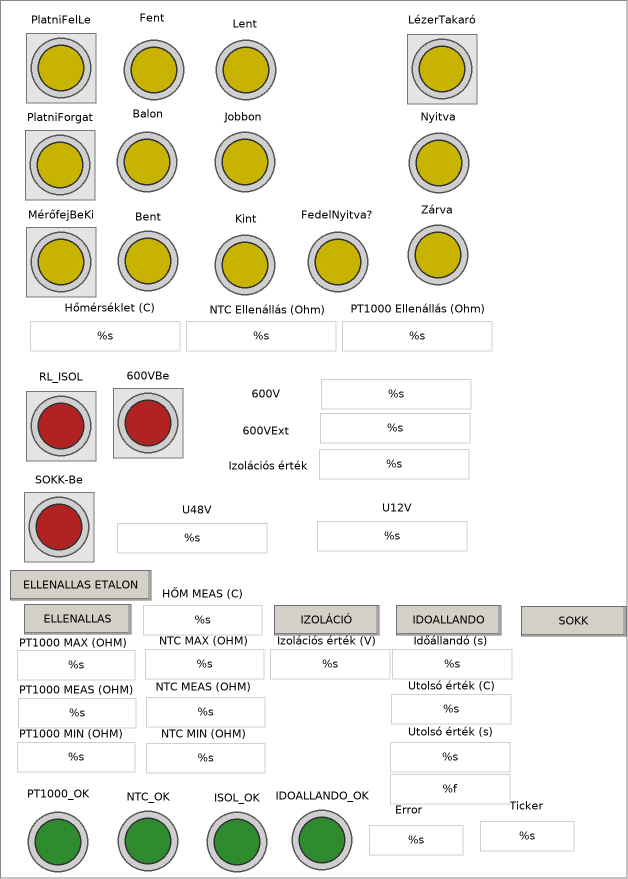
VISUALIZATION TempPistiVegmero  // 628x879
    Lamp1 (211,35 70x70), variable: VEGMERO.bPlatniLent, style: Lamp-Lamp1-Yellow
    Label (190,9 110x30), "Lent"
    PushSwitch (26,33 70x70), variable: VEGMERO.bPlatniFelLe, behaviour: TOGGLE, style: Switch-PushSwitch-Yellow
    Label (6,5 110x30), "PlatniFelLe"
    Lamp1 (112,127 70x70), variable: VEGMERO.bPlatniBalon, style: Lamp-Lamp1-Yellow
    Label (93,99 110x30), "Balon"
    Lamp1 (210,127 70x70), variable: VEGMERO.bPlatniJobbon, style: Lamp-Lamp1-Yellow
    Label (188,102 110x30), "Jobbon"
    PushSwitch (25,130 70x70), variable: VEGMERO.bPlatniBalraJobbra, behaviour: TOGGLE, style: Switch-PushSwitch-Yellow
    Label (5,103 110x29), "PlatniForgat"
    Lamp1 (113,226 70x70), variable: VEGMERO.bMerotukBent, style: Lamp-Lamp1-Yellow
    Label (93,202 110x30), "Bent"
    Lamp1 (210,230 70x70), variable: VEGMERO.bMerotukKint, style: Lamp-Lamp1-Yellow
    Label (191,204 110x30), "Kint"
    PushSwitch (26,227 70x70), variable: VEGMERO.bMerotukBeKi, behaviour: TOGGLE, style: Switch-PushSwitch-Yellow
    Label (6,200 110x30), "MérőfejBeKi"
    Lamp1 (119,35 70x70), variable: VEGMERO.bPlatniFent, style: Lamp-Lamp1-Yellow
    Label (97,3 110x30), "Fent"
    Lamp1 (303,227 70x70), variable: VEGMERO.bFedelNyitva, style: Lamp-Lamp1-Yellow
    Label (282,200 110x30), "FedelNyitva?"
    PushSwitch (26,391 70x70), variable: VEGMERO.bRL_ISOL, behaviour: TOGGLE, style: Switch-PushSwitch-Red
    Label (6,362 110x30), "RL_ISOL"
    Textfield (321,379 150x30), "%s", text variable: VEGMERO.U600V_TRANS, input disabled if: TRUE
    Textfield (186,321 150x30), "%s", text variable: VEGMERO.NTRES_CALC, input disabled if: TRUE
    Textfield (342,321 150x30), "%s", text variable: VEGMERO.PTRES_CALC, input disabled if: TRUE
    Label (207,295 121x30), "NTC Ellenállás (Ohm)"
    Label (347,294 142x30), "PT1000 Ellenállás (Ohm)"
    Label (211,379 110x30), "600V"
    PushSwitch (113,388 70x70), variable: VEGMERO.b600VBe, behaviour: TOGGLE, style: Switch-PushSwitch-Red
    Label (93,361 110x30), "600VBe"
    Textfield (117,523 150x30), "%s", text variable: VEGMERO.U48V_TRANS, input disabled if: TRUE
    Label (142,495 110x30), "U48V"
    Textfield (320,413 150x30), "%s", text variable: VEGMERO.U600VExt_TRANS, input disabled if: TRUE
    Label (211,416 110x30), "600VExt"
    Textfield (319,449 150x30), "%s", text variable: VEGMERO.UISOL_TRANS, input disabled if: TRUE
    Label (213,451 110x30), "Izolációs érték"
    PushSwitch (24,492 70x70), variable: VEGMERO.PT_SOKK48V, behaviour: TOGGLE, style: Switch-PushSwitch-Red
    Label (4,465 110x30), "SOKK-Be"
    Textfield (317,521 150x30), "%s", text variable: VEGMERO.U12V_TRANS, input disabled if: TRUE
    Label (342,493 110x30), "U12V"
    Lamp1 (23,807 70x70), variable: VEGMERO.bPTRES_OK, style: Lamp-Lamp1-Green
    Label (4,750 110x30), "PT1000_OK"
    Lamp1 (113,806 70x70), variable: VEGMERO.bNTCRES_OK, style: Lamp-Lamp1-Green
    Label (93,782 110x30), "NTC_OK"
    Textfield (30,321 150x30), "%s", text variable: VEGMERO.rHoerzekelo_TRANS, input disabled if: TRUE
    Label (55,293 110x30), "Hőmérséklet (C)"
    Lamp1 (202,807 70x70), variable: VEGMERO.bISOL_OK, style: Lamp-Lamp1-Green
    Label (182,783 110x30), "ISOL_OK"
    Button (24,604 107x30), "ELLENALLAS", input disabled if: VEGMERO.s_InCommand<>''
        OnMouseUp: execute { VEGMERO.s_InCommand:='ELLENALLAS'; }
    Button (274,605 105x30), "IZOLÁCIÓ", input disabled if: VEGMERO.s_InCommand<>''
        OnMouseUp: execute { VEGMERO.s_InCommand:='ATUTES'; }
    Textfield (18,698 118x30), "%s", text variable: VEGMERO.rPTRES, input disabled if: TRUE
    Textfield (146,697 119x30), "%s", text variable: VEGMERO.rNTCRES, input disabled if: TRUE
    Textfield (270,649 120x30), "%s", text variable: VEGMERO.rISOL, input disabled if: TRUE
    Textfield (369,825 94x30), "%s", text variable: VEGMERO.n_OutErrId, input disabled if: TRUE
    Textfield (17,742 118x30), "%s", text variable: VEGMERO.PTRES_MIN, input disabled if: TRUE
    Textfield (17,650 118x30), "%s", text variable: VEGMERO.PTRES_MAX, input disabled if: TRUE
    Textfield (146,743 119x30), "%s", text variable: VEGMERO.NTCRES_MIN, input disabled if: TRUE
    Textfield (145,649 119x30), "%s", text variable: VEGMERO.NTCRES_MAX, input disabled if: TRUE
    Textfield (143,605 119x30), "%s", text variable: VEGMERO.rTemp, input disabled if: TRUE
    Button (396,605 105x30), "IDOALLANDO", input disabled if: VEGMERO.s_InCommand<>''
        OnMouseUp: execute { VEGMERO.s_InCommand:='IDOALLANDO'; }
    Textfield (392,649 120x30), "%s", text variable: VEGMERO.tIdoallando, input disabled if: TRUE
    Textfield (391,694 120x30), "%s", text variable: VEGMERO.arIdoallandoPTTEMP[VEGMERO.nI], input disabled if: TRUE
    Textfield (390,742 120x30), "%s", text variable: VEGMERO.atIdoallando[VEGMERO.nI], input disabled if: TRUE
    Label (16,719 110x30), "PT1000 MIN (OHM)"
    Label (18,675 117x30), "PT1000 MEAS (OHM)"
    Label (18,628 110x30), "PT1000 MAX (OHM)"
    Label (132,626 143x30), "NTC MAX (OHM)"
    Label (132,719 143x30), "NTC MIN (OHM)"
    Label (132,672 143x30), "NTC MEAS (OHM)"
    Label (255,626 143x30), "Izolációs érték (V)"
    Label (131,579 143x30), "HŐM MEAS (C)"
    Label (379,626 143x30), "Időállandó (s)"
    Label (380,671 143x30), "Utolsó érték (C)"
    Label (379,717 143x30), "Utolsó érték (s)"
    Label (337,795 143x30), "Error"
    Button (521,606 105x30), "SOKK", input disabled if: VEGMERO.s_InCommand<>''
        OnMouseUp: execute { VEGMERO.s_InCommand:='SOKK'; }
    Textfield (480,821 94x30), "%s", text variable: VEGMERO.tTickerET, input disabled if: TRUE
    Label (455,791 143x30), "Ticker"
    Lamp1 (287,805 70x70), variable: VEGMERO.bIDOALLANDO_OK, style: Lamp-Lamp1-Green
    Label (267,781 110x30), "IDOALLANDO_OK"
    Textfield (390,774 120x30), "%f", text variable: GVL.rTempMax
        OnMouseClick: write the text variable via VisuDialogs.Numpad, min 0, max 400
    Button (10,570 141x30), "ELLENALLAS ETALON", input disabled if: VEGMERO.s_InCommand<>''
        OnMouseUp: execute { VEGMERO.s_InCommand:='ELLENALLASETALON'; }
    Label (3,779 110x30), "PT1000_OK"
    PushSwitch (407,34 70x70), variable: VEGMERO.bLezertakaro, behaviour: TOGGLE, style: Switch-PushSwitch-Yellow
    Label (387,5 110x30), "LézerTakaró"
    Lamp1 (404,128 70x70), variable: VEGMERO.bLezertakaroNyitva, style: Lamp-Lamp1-Yellow
    Label (383,102 110x30), "Nyitva"
    Lamp1 (403,220 70x70), variable: VEGMERO.bLezertakaroZarva, style: Lamp-Lamp1-Yellow
    Label (382,195 110x30), "Zárva"
END_VISUALIZATION

(* stored: Version 1.1.0.1, ProductVersion 3.1.4024.11
   Visu TempPistiVegmero: Id {5fd14475-ff2f-4515-9b0f-7359e1c2c478} *)
